Universal Robots PolyScope program: wait_program.urp

Program wait_program (installation=default directory=/ursim/programs createdIn=3.15.8.106339 lastSavedIn=3.12.1.90940 robotSerialNumber=2018359999)
Calibrated DH parameters: a=[0, -0.425, -0.39225, 0, 0, 0]; d=[0.089159, 0, 0, 0.10915, 0.09465, 0.0823]; alpha=[1.570796, 0, 0, 1.570796, -1.570796, 0]; deltaTheta=[0, 0, 0, 0, 0, 0]
Robot Program (runOnlyOnce=false)
  Wait Sleep waitTime=0.01
